Yaskawa INFORM job: MALBEN2.JBI

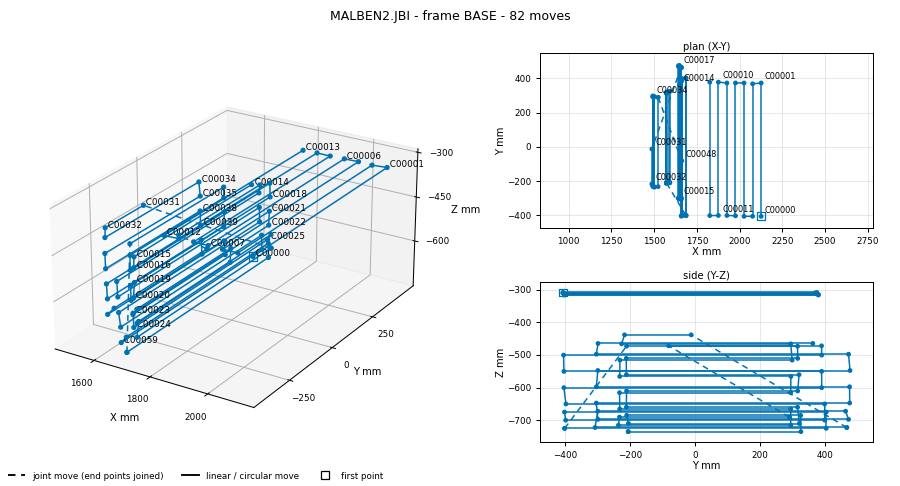
[picture p0: tool path of MALBEN2.JBI in frame BASE, 82 of 88 moves have a stored position in this frame; points joined in program order, loops and branches not executed]
/JOB
//NAME MALBEN2
//POS
///NPOS 82,0,82,0,0,0
///TOOL 0
///POSTYPE BASE
///RECTAN
///RCONF 1,0,0,0,0,0,0,0,0,0,0,0,0,0,0,0,0,0,0,0,0,0,0,0
C00000=2125.909445,-406.008973,-308.104381,175.000000,5.000000,5.000000
C00001=2125.909445,373.660402,-308.104381,175.000000,5.000000,5.000000
C00002=2075.909445,368.819494,-309.393068,175.000000,5.000000,5.000000
C00003=2075.909445,-405.716187,-309.393068,175.000000,5.000000,5.000000
C00004=2025.909445,-405.951122,-310.182147,175.000000,5.000000,5.000000
C00005=2025.909445,373.660402,-310.182147,175.000000,5.000000,5.000000
C00006=1975.909445,373.956280,-311.477162,175.000000,5.000000,5.000000
C00007=1975.909445,-402.823433,-311.477162,175.000000,5.000000,5.000000
C00008=1925.909445,-400.874837,-312.665221,175.000000,5.000000,5.000000
C00009=1925.909445,373.660402,-312.665221,175.000000,5.000000,5.000000
C00010=1875.909445,378.502193,-314.362338,175.000000,5.000000,5.000000
C00011=1875.909445,-400.874837,-314.362338,175.000000,5.000000,5.000000
C00012=1825.577046,-401.602166,-315.947729,175.000000,5.000000,5.000000
C00013=1825.577046,378.502193,-315.947729,175.000000,5.000000,5.000000
C00014=1647.531093,361.329041,-464.681952,175.000000,-89.999999,5.000000
C00015=1647.531093,-298.349229,-464.681952,175.000000,-89.999999,5.000000
C00016=1649.095223,-303.404759,-497.748608,175.000000,-89.999999,5.000000
C00017=1649.095223,471.072188,-497.748608,175.000000,-89.999999,5.000000
C00018=1647.785777,475.683018,-547.748608,175.000000,-89.999999,5.000000
C00019=1647.785777,-298.944959,-547.748608,175.000000,-89.999999,5.000000
C00020=1646.019881,-303.463051,-597.748608,175.000000,-89.999999,5.000000
C00021=1646.019881,474.299902,-597.748608,175.000000,-89.999999,5.000000
C00022=1643.806967,474.620068,-647.748608,175.000000,-89.999999,5.000000
C00023=1643.806967,-303.703286,-647.748608,175.000000,-89.999999,5.000000
C00024=1641.764926,-298.622143,-697.748608,175.000000,-89.999999,5.000000
C00025=1641.764926,471.072188,-697.748608,175.000000,-89.999999,5.000000
C00026=1660.154489,461.999791,-672.748608,180.000000,-60.000000,0.000000
C00027=1660.154489,-298.944959,-672.748608,180.000000,-60.000000,0.000000
C00028=1658.630608,-307.498024,-722.748608,180.000000,-60.000000,0.000000
C00029=1658.630608,465.692077,-722.748608,180.000000,-60.000000,0.000000
C00030=1658.630608,465.692077,-722.748608,180.000000,-60.000000,0.000000
C00031=1487.056680,-12.244425,-438.225594,175.000000,-89.999999,5.000000
C00032=1487.056680,-216.807296,-438.225594,175.000000,-89.999999,5.000000
C00033=1491.788510,-225.939630,-465.851344,175.000000,-89.999999,5.000000
C00034=1491.788510,293.594004,-465.851344,175.000000,-89.999999,5.000000
C00035=1493.706990,297.926988,-515.851344,175.000000,-89.999999,5.000000
C00036=1493.706990,-231.071040,-515.851344,175.000000,-89.999999,5.000000
C00037=1495.372210,-231.643974,-565.851344,175.000000,-89.999999,5.000000
C00038=1495.372210,293.974678,-565.851344,175.000000,-89.999999,5.000000
C00039=1497.290733,293.592082,-615.851344,175.000000,-89.999999,5.000000
C00040=1497.290733,-232.212239,-615.851344,175.000000,-89.999999,5.000000
C00041=1499.126097,-231.645347,-665.851344,175.000000,-89.999999,5.000000
C00042=1499.126097,293.592356,-665.851344,175.000000,-89.999999,5.000000
C00043=1501.346927,293.591395,-715.851344,175.000000,-89.999999,5.000000
C00044=1501.346927,-235.692413,-715.851344,175.000000,-89.999999,5.000000
C00045=1523.655226,-232.314411,-690.851344,180.000000,-60.000000,0.000000
C00046=1523.655226,289.408511,-690.851344,180.000000,-60.000000,0.000000
C00047=1523.655226,289.408511,-690.851344,180.000000,-60.000000,0.000000
C00048=1662.229022,-81.378205,-471.863635,175.000000,-89.999999,5.000000
C00049=1662.229022,388.136901,-471.863635,175.000000,-89.999999,5.000000
C00050=1658.564852,388.674780,-500.419594,175.000000,-89.999999,5.000000
C00051=1658.564852,-404.150984,-500.419594,175.000000,-89.999999,5.000000
C00052=1660.302756,-403.074785,-550.419594,175.000000,-89.999999,5.000000
C00053=1660.302756,388.459717,-550.419594,175.000000,-89.999999,5.000000
C00054=1661.970730,388.674780,-600.419594,175.000000,-89.999999,5.000000
C00055=1661.970730,-403.228906,-600.419594,175.000000,-89.999999,5.000000
C00056=1663.500978,-396.888297,-650.419594,175.000000,-89.999999,5.000000
C00057=1663.500978,397.820042,-650.419594,175.000000,-89.999999,5.000000
C00058=1664.833382,398.142858,-700.419594,175.000000,-89.999999,5.000000
C00059=1664.833382,-397.695115,-700.419594,175.000000,-89.999999,5.000000
C00060=1686.014757,-401.289805,-675.419594,180.000000,-60.000000,0.000000
C00061=1686.014757,402.661834,-675.419594,180.000000,-60.000000,0.000000
C00062=1686.688388,402.661834,-725.419594,180.000000,-60.000000,0.000000
C00063=1686.688388,-400.922828,-725.419594,180.000000,-60.000000,0.000000
C00064=1686.688388,-400.922828,-725.419594,180.000000,-60.000000,0.000000
C00065=1572.281953,-210.681608,-473.110843,175.000000,-89.999999,5.000000
C00066=1572.281953,314.551427,-473.110843,175.000000,-89.999999,5.000000
C00067=1572.150400,314.931826,-510.561428,175.000000,-89.999999,5.000000
C00068=1572.150400,-211.592369,-510.561428,175.000000,-89.999999,5.000000
C00069=1571.863689,-211.135890,-560.561428,175.000000,-89.999999,5.000000
C00070=1571.863689,319.118967,-560.561428,175.000000,-89.999999,5.000000
C00071=1571.523786,314.935397,-610.561428,175.000000,-89.999999,5.000000
C00072=1571.523786,-210.682981,-610.561428,175.000000,-89.999999,5.000000
C00073=1572.417463,-211.293955,-660.561428,175.000000,-89.999999,5.000000
C00074=1572.417463,314.554448,-660.561428,175.000000,-89.999999,5.000000
C00075=1573.818584,319.891027,-710.561428,175.000000,-89.999999,5.000000
C00076=1573.818584,-204.976989,-710.561428,175.000000,-89.999999,5.000000
C00077=1592.515603,-210.305603,-685.561428,180.000000,-60.000000,0.000000
C00078=1592.515603,324.073224,-685.561428,180.000000,-60.000000,0.000000
C00079=1589.870735,324.691476,-735.561428,180.000000,-60.000000,0.000000
C00080=1589.870735,-205.627925,-735.561428,180.000000,-60.000000,0.000000
C00081=1589.870735,-205.627925,-735.561428,180.000000,-60.000000,0.000000
///POSTYPE PULSE
///PULSE
EC00000=0
EC00001=0
EC00002=0
EC00003=0
EC00004=0
EC00005=0
EC00006=0
EC00007=0
EC00008=0
EC00009=0
EC00010=0
EC00011=0
EC00012=0
EC00013=0
EC00014=0
EC00015=0
EC00016=0
EC00017=0
EC00018=0
EC00019=0
EC00020=0
EC00021=0
EC00022=0
EC00023=0
EC00024=0
EC00025=0
EC00026=0
EC00027=0
EC00028=0
EC00029=0
EC00030=92160
EC00031=92160
EC00032=92160
EC00033=92160
EC00034=92160
EC00035=92160
EC00036=92160
EC00037=92160
EC00038=92160
EC00039=92160
EC00040=92160
EC00041=92160
EC00042=92160
EC00043=92160
EC00044=92160
EC00045=92160
EC00046=92160
EC00047=184320
EC00048=184320
EC00049=184320
EC00050=184320
EC00051=184320
EC00052=184320
EC00053=184320
EC00054=184320
EC00055=184320
EC00056=184320
EC00057=184320
EC00058=184320
EC00059=184320
EC00060=184320
EC00061=184320
EC00062=184320
EC00063=184320
EC00064=276480
EC00065=276480
EC00066=276480
EC00067=276480
EC00068=276480
EC00069=276480
EC00070=276480
EC00071=276480
EC00072=276480
EC00073=276480
EC00074=276480
EC00075=276480
EC00076=276480
EC00077=276480
EC00078=276480
EC00079=276480
EC00080=276480
EC00081=368640
//INST
///DATE 2023/02/07 12:30
///ATTR SC,RW,RJ
////FRAME BASE
///GROUP1 RB1,ST1
NOP
MOVJ P009 EX000 VJ=15.00
MOVJ C00000 EC00000 VJ=15.0
CALL JOB:SPYON
MOVL C00001 EC00001 V=150.0
MOVL C00002 EC00002 V=150.0
MOVL C00003 EC00003 V=150.0
MOVL C00004 EC00004 V=150.0
MOVL C00005 EC00005 V=150.0
MOVL C00006 EC00006 V=150.0
MOVL C00007 EC00007 V=150.0
MOVL C00008 EC00008 V=150.0
MOVL C00009 EC00009 V=150.0
MOVL C00010 EC00010 V=150.0
MOVL C00011 EC00011 V=150.0
MOVL C00012 EC00012 V=150.0
MOVL C00013 EC00013 V=150.0
CALL JOB:SPYOF
MOVJ P009 VJ=15.00
MOVJ C00014 EC00014 VJ=15.0
CALL JOB:SPYON
MOVL C00015 EC00015 V=150.0
MOVL C00016 EC00016 V=150.0
MOVL C00017 EC00017 V=150.0
MOVL C00018 EC00018 V=150.0
MOVL C00019 EC00019 V=150.0
MOVL C00020 EC00020 V=150.0
MOVL C00021 EC00021 V=150.0
MOVL C00022 EC00022 V=150.0
MOVL C00023 EC00023 V=150.0
MOVL C00024 EC00024 V=150.0
MOVL C00025 EC00025 V=150.0
MOVL C00026 EC00026 V=150.0
MOVL C00027 EC00027 V=150.0
MOVL C00028 EC00028 V=150.0
MOVL C00029 EC00029 V=150.0
CALL JOB:SPYOF
MOVJ P009 VJ=15.00
MOVL C00030 EC00030 V=150.0
MOVJ C00031 EC00031 VJ=15.0
CALL JOB:SPYON
MOVL C00032 EC00032 V=150.0
MOVL C00033 EC00033 V=150.0
MOVL C00034 EC00034 V=150.0
MOVL C00035 EC00035 V=150.0
MOVL C00036 EC00036 V=150.0
MOVL C00037 EC00037 V=150.0
MOVL C00038 EC00038 V=150.0
MOVL C00039 EC00039 V=150.0
MOVL C00040 EC00040 V=150.0
MOVL C00041 EC00041 V=150.0
MOVL C00042 EC00042 V=150.0
MOVL C00043 EC00043 V=150.0
MOVL C00044 EC00044 V=150.0
MOVL C00045 EC00045 V=150.0
MOVL C00046 EC00046 V=150.0
CALL JOB:SPYOF
MOVJ P009 VJ=15.00
MOVL C00047 EC00047 V=150.0
MOVJ C00048 EC00048 VJ=15.0
CALL JOB:SPYON
MOVL C00049 EC00049 V=150.0
MOVL C00050 EC00050 V=150.0
MOVL C00051 EC00051 V=150.0
MOVL C00052 EC00052 V=150.0
MOVL C00053 EC00053 V=150.0
MOVL C00054 EC00054 V=150.0
MOVL C00055 EC00055 V=150.0
MOVL C00056 EC00056 V=150.0
MOVL C00057 EC00057 V=150.0
MOVL C00058 EC00058 V=150.0
MOVL C00059 EC00059 V=150.0
MOVL C00060 EC00060 V=150.0
MOVL C00061 EC00061 V=150.0
MOVL C00062 EC00062 V=150.0
MOVL C00063 EC00063 V=150.0
CALL JOB:SPYOF
MOVJ P009 VJ=15.00
MOVL C00064 EC00064 V=150.0
MOVJ C00065 EC00065 VJ=15.0
CALL JOB:SPYON
MOVL C00066 EC00066 V=150.0
MOVL C00067 EC00067 V=150.0
MOVL C00068 EC00068 V=150.0
MOVL C00069 EC00069 V=150.0
MOVL C00070 EC00070 V=150.0
MOVL C00071 EC00071 V=150.0
MOVL C00072 EC00072 V=150.0
MOVL C00073 EC00073 V=150.0
MOVL C00074 EC00074 V=150.0
MOVL C00075 EC00075 V=150.0
MOVL C00076 EC00076 V=150.0
MOVL C00077 EC00077 V=150.0
MOVL C00078 EC00078 V=150.0
MOVL C00079 EC00079 V=150.0
MOVL C00080 EC00080 V=150.0
CALL JOB:SPYOF
MOVJ P009 VJ=15.00
MOVL C00081 EC00081 V=150.0
END
